// Brief: Setup Arm Move to Package Posture
FUNCTION_BLOCK PUBLIC FB_SetupCtrlPackage EXTENDS FB_SetupArmCtrlBase
VAR_INPUT
END_VAR
VAR_OUTPUT
END_VAR
VAR
END_VAR

METHOD PUBLIC init : BOOL
VAR_IN_OUT CONSTANT
	i_setupArm	:FB_SetupArm;
END_VAR
VAR_IN_OUT 
	r_setupArmCtrlCmd :ST_SetupArmCtrlCmds;
END_VAR
SUPER^.Init(i_setupArm,r_setupArmCtrlCmd);
END_METHOD

END_FUNCTION_BLOCK

(* stored: Version 1.1.0.1, ProductVersion 3.1.4024.12
   POU FB_SetupCtrlPackage: Id {3caa7d81-2fc0-4b44-8421-fc376f3615bb}, SpecialFunc None
   Method init: Id {2d8c4ce8-f95d-44ef-b5b3-99ca1edcf8a1} *)
